// Mitsubishi GX Works2 project: Final Project(24.06.05)   PLC: Q00U

PROGRAM CLDa
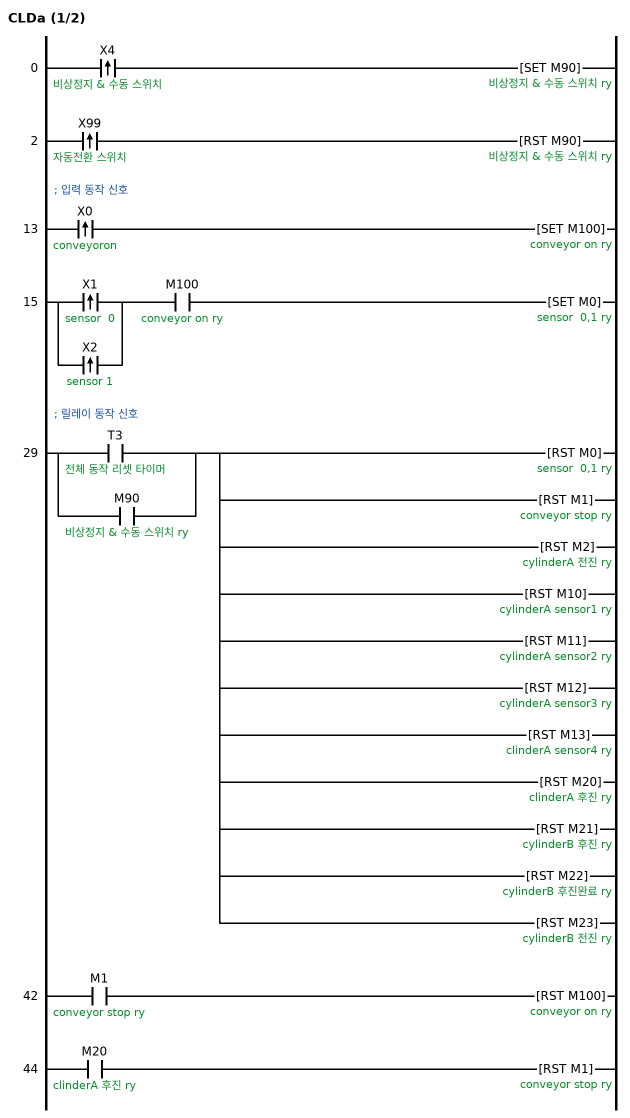
0     LDP     X4  ; 비상정지 & 수동 스위치
      SET     M90  ; 비상정지 & 수동 스위치 ry
2     LDP     X99  ; 자동전환 스위치
      RST     M90  ; 비상정지 & 수동 스위치 ry
; 입력 동작 신호
13    LDP     X0  ; conveyoron
      SET     M100  ; conveyor on ry
15    LDP     X1  ; sensor  0
      ORP     X2  ; sensor 1
      AND     M100  ; conveyor on ry
      SET     M0  ; sensor  0,1 ry
; 릴레이 동작 신호
29    LD      T3  ; 전체 동작 리셋 타이머
      OR      M90  ; 비상정지 & 수동 스위치 ry
      RST     M0  ; sensor  0,1 ry
      RST     M1  ; conveyor stop ry
      RST     M2  ; cylinderA 전진 ry
      RST     M10  ; cylinderA sensor1 ry
      RST     M11  ; cylinderA sensor2 ry
      RST     M12  ; cylinderA sensor3 ry
      RST     M13  ; clinderA sensor4 ry
      RST     M20  ; clinderA 후진 ry
      RST     M21  ; cylinderB 후진 ry
      RST     M22  ; cylinderB 후진완료 ry
      RST     M23  ; cylinderB 전진 ry
42    LD      M1  ; conveyor stop ry
      RST     M100  ; conveyor on ry
44    LD      M20  ; clinderA 후진 ry
      RST     M1  ; conveyor stop ry
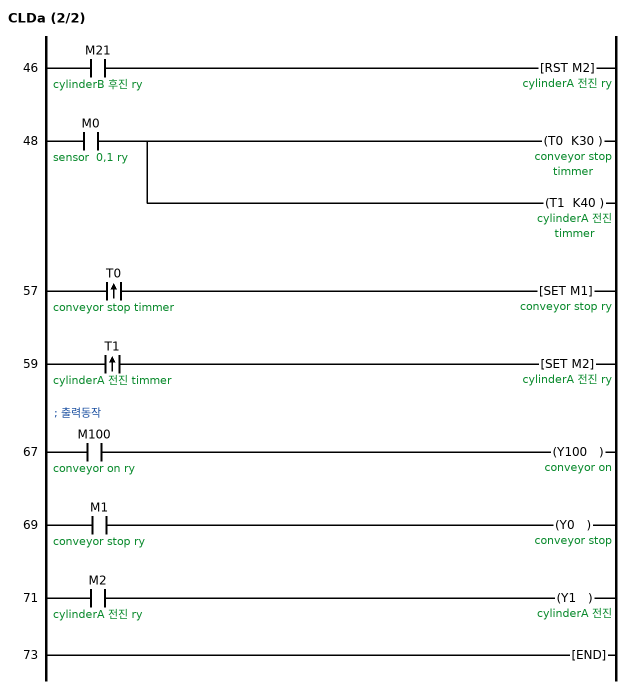
46    LD      M21  ; cylinderB 후진 ry
      RST     M2  ; cylinderA 전진 ry
48    LD      M0  ; sensor  0,1 ry
      OUT     T0 K30  ; conveyor stop timmer
      OUT     T1 K40  ; cylinderA 전진 timmer
57    LDP     T0  ; conveyor stop timmer
      SET     M1  ; conveyor stop ry
59    LDP     T1  ; cylinderA 전진 timmer
      SET     M2  ; cylinderA 전진 ry
; 출력동작
67    LD      M100  ; conveyor on ry
      OUT     Y100  ; conveyor on
69    LD      M1  ; conveyor stop ry
      OUT     Y0  ; conveyor stop
71    LD      M2  ; cylinderA 전진 ry
      OUT     Y1  ; cylinderA 전진
73    END
END_PROGRAM

PROGRAM sensor1
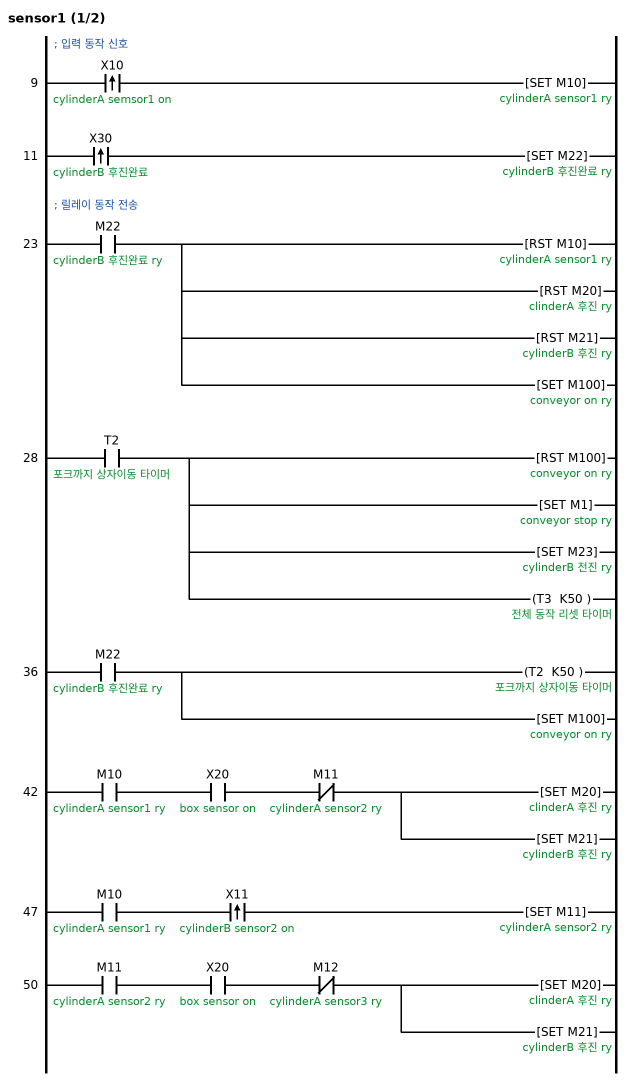
; 입력 동작 신호
9     LDP     X10  ; cylinderA semsor1 on
      SET     M10  ; cylinderA sensor1 ry
11    LDP     X30  ; cylinderB 후진완료
      SET     M22  ; cylinderB 후진완료 ry
; 릴레이 동작 전송
23    LD      M22  ; cylinderB 후진완료 ry
      RST     M10  ; cylinderA sensor1 ry
      RST     M20  ; clinderA 후진 ry
      RST     M21  ; cylinderB 후진 ry
      SET     M100  ; conveyor on ry
28    LD      T2  ; 포크까지 상자이동 타이머
      RST     M100  ; conveyor on ry
      SET     M1  ; conveyor stop ry
      SET     M23  ; cylinderB 전진 ry
      OUT     T3 K50  ; 전체 동작 리셋 타이머
36    LD      M22  ; cylinderB 후진완료 ry
      OUT     T2 K50  ; 포크까지 상자이동 타이머
      SET     M100  ; conveyor on ry
42    LD      M10  ; cylinderA sensor1 ry
      AND     X20  ; box sensor on
      ANI     M11  ; cylinderA sensor2 ry
      SET     M20  ; clinderA 후진 ry
      SET     M21  ; cylinderB 후진 ry
47    LD      M10  ; cylinderA sensor1 ry
      ANDP    X11  ; cylinderB sensor2 on
      SET     M11  ; cylinderA sensor2 ry
50    LD      M11  ; cylinderA sensor2 ry
      AND     X20  ; box sensor on
      ANI     M12  ; cylinderA sensor3 ry
      SET     M20  ; clinderA 후진 ry
      SET     M21  ; cylinderB 후진 ry
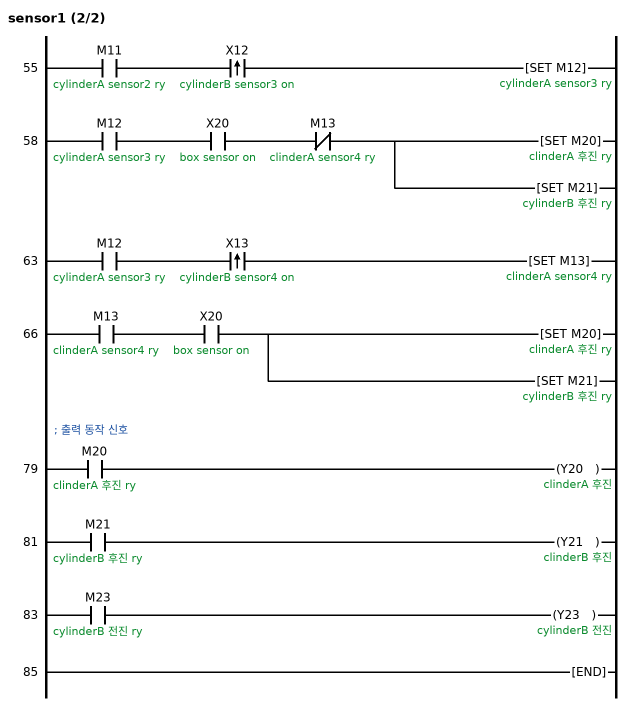
55    LD      M11  ; cylinderA sensor2 ry
      ANDP    X12  ; cylinderB sensor3 on
      SET     M12  ; cylinderA sensor3 ry
58    LD      M12  ; cylinderA sensor3 ry
      AND     X20  ; box sensor on
      ANI     M13  ; clinderA sensor4 ry
      SET     M20  ; clinderA 후진 ry
      SET     M21  ; cylinderB 후진 ry
63    LD      M12  ; cylinderA sensor3 ry
      ANDP    X13  ; cylinderB sensor4 on
      SET     M13  ; clinderA sensor4 ry
66    LD      M13  ; clinderA sensor4 ry
      AND     X20  ; box sensor on
      SET     M20  ; clinderA 후진 ry
      SET     M21  ; cylinderB 후진 ry
; 출력 동작 신호
79    LD      M20  ; clinderA 후진 ry
      OUT     Y20  ; clinderA 후진
81    LD      M21  ; cylinderB 후진 ry
      OUT     Y21  ; clinderB 후진
83    LD      M23  ; cylinderB 전진 ry
      OUT     Y23  ; cylinderB 전진
85    END
END_PROGRAM

PROGRAM M10
0     END
END_PROGRAM

PROGRAM manual
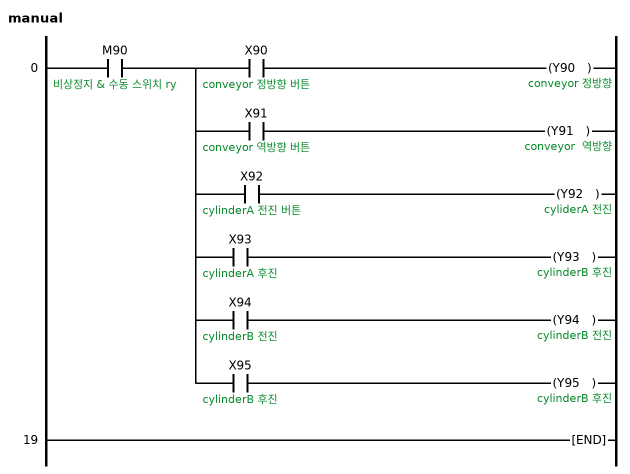
0     LD      M90  ; 비상정지 & 수동 스위치 ry
      MPS
      AND     X90  ; conveyor 정방향 버튼
      OUT     Y90  ; conveyor 정방향
      MRD
      AND     X91  ; conveyor 역방향 버튼
      OUT     Y91  ; conveyor  역방향
      MRD
      AND     X92  ; cylinderA 전진 버튼
      OUT     Y92  ; cyliderA 전진
      MRD
      AND     X93  ; cylinderA 후진
      OUT     Y93  ; cylinderB 후진
      MRD
      AND     X94  ; cylinderB 전진
      OUT     Y94  ; cylinderB 전진
      MPP
      AND     X95  ; cylinderB 후진
      OUT     Y95  ; cylinderB 후진
19    END
END_PROGRAM

// device comments not shown above
X80  ; 자동 스위치
